ABB RobotStudio station: LATAM_caja_negra.rsstnx

Station Project3 (saved by RobotStudio 23.2.10395.0)
Controller IRB6640_130_320, task T_ROB1: task frame (RAPID world) sits at (1140.52, 0, 0) mm in the station
Controller IRB6640_130_320
  mechanical unit ROB_1: IRB6640_130_320__04, 6 joints, base frame (0, 0, 0) mm
Layout (positions relative to the parent item):
  - IRB6640_130_320__04 [mechanism, from %ABB.RobotStudio.Models.IRB6640%\IRB6640_130_320_G_04.rslib] at (1140.52, 0, 0) mm; joint values [0, 0, 0, 0, 0.1599, 0.0179] (rad or m)
  - Grupo_2 [graphiccomponentgroup]
    - Euro Pallet [graphiccomponentgroup, from Equipment\Euro Pallet.rslib] at (0, -2846.4, -3.2) mm
      - Body 1 [part, from Equipment\Euro Pallet.rslib]
    - Euro Pallet_2 [graphiccomponentgroup, from Equipment\Euro Pallet.rslib] at (0, -2029.21, -3.2) mm
      - Body 1 [part, from Equipment\Euro Pallet.rslib]
    - Euro Pallet_4 [graphiccomponentgroup, from Equipment\Euro Pallet.rslib] at (1157.68, -2846.4, -3.2) mm
      - Body 1 [part, from Equipment\Euro Pallet.rslib]
    - Euro Pallet_3 [graphiccomponentgroup, from Equipment\Euro Pallet.rslib] at (1157.68, -2029.21, -3.2) mm
      - Body 1 [part, from Equipment\Euro Pallet.rslib]
  - IRC5 [part, from %ABB.RobotStudio.Models.IRC5%\IRC5_Control-Module.rslib] at (5669.92, -980.14, 100) mm, rotated rx 90 ry 0 rz 90 deg
  - Pieza_2 [part] at (1194.52, -1963.54, 134.82) mm, size 600 x 600 x 200 mm
  - propeller [part, from Training Objects\propeller.rslib] at (625, 0, 373) mm, rotated rx 0 ry 0 rz 12 deg
  - IRB1200_5_90_STD_03 [mechanism, from %ABB.RobotStudio.Models.IRB1200%\IRB1200_5_90_STD_03.rslib] at (3914.45, 3690.17, 640.27) mm, rotated rx 0 ry 0 rz -177.61 deg; joint values [0, 0, 0, 0, 0.5236, 0] (rad or m)
  - Pieza_3 [part] at (3715.49, 3430.98, 0) mm, size 500 x 500 x 600 mm
  - Grupo_3 [graphiccomponentgroup]
    - Fence_2500_3 [graphiccomponentgroup, from Equipment\Fence_2500.rslib] at (-6063.8, 1734.17, 0) mm
      - Body 1 [part, from Equipment\Fence_2500.rslib]
      - Body 2 [part, from Equipment\Fence_2500.rslib]
    - Fence_2500_4 [graphiccomponentgroup, from Equipment\Fence_2500.rslib] at (-5999.52, 4213.05, 0) mm
      - Body 1 [part, from Equipment\Fence_2500.rslib]
      - Body 2 [part, from Equipment\Fence_2500.rslib]
    - Fence_2500_2 [graphiccomponentgroup, from Equipment\Fence_2500.rslib] at (-6042.58, -669.32, 0) mm
      - Body 1 [part, from Equipment\Fence_2500.rslib] at (0, -91.47, 0) mm
      - Body 2 [part, from Equipment\Fence_2500.rslib]
    - Fence_2500 [graphiccomponentgroup, from Equipment\Fence_2500.rslib] at (-5950.27, -3103.88, 0) mm
      - Body 1 [part, from Equipment\Fence_2500.rslib] at (0, -91.47, 0) mm
      - Body 2 [part, from Equipment\Fence_2500.rslib]
  - Grupo_4 [graphiccomponentgroup] at (10944.14, 0, 0) mm
    - Fence_2500_3 [graphiccomponentgroup, from Equipment\Fence_2500.rslib] at (-6063.8, 1734.17, 0) mm
      - Body 1 [part, from Equipment\Fence_2500.rslib]
      - Body 2 [part, from Equipment\Fence_2500.rslib]
    - Fence_2500_4 [graphiccomponentgroup, from Equipment\Fence_2500.rslib] at (-5999.52, 4213.05, 0) mm
      - Body 1 [part, from Equipment\Fence_2500.rslib]
      - Body 2 [part, from Equipment\Fence_2500.rslib]
    - Fence_2500_2 [graphiccomponentgroup, from Equipment\Fence_2500.rslib] at (-6042.58, -669.32, 0) mm
      - Body 1 [part, from Equipment\Fence_2500.rslib] at (0, -91.47, 0) mm
      - Body 2 [part, from Equipment\Fence_2500.rslib]
    - Fence_2500 [graphiccomponentgroup, from Equipment\Fence_2500.rslib] at (-5950.27, -3103.88, 0) mm
      - Body 1 [part, from Equipment\Fence_2500.rslib] at (0, -91.47, 0) mm
      - Body 2 [part, from Equipment\Fence_2500.rslib]
  - Grupo_5 [graphiccomponentgroup]
    - 950_4000_h2 [part, from %ABB.RobotStudio.Models.Conveyors%\Conveyor 950 4000 h2.rslib] at (3638.72, -1101.13, 242.49) mm, rotated rx 0 ry 0 rz 90.05 deg
    - 950_4000 [part, from %ABB.RobotStudio.Models.Conveyors%\Conveyor 950 4000 h2.rslib] at (3638.72, 3166.35, 242.49) mm, rotated rx 0 ry 0 rz 90.05 deg
  - Grupo_6 [graphiccomponentgroup] at (0, -9897.8, 0) mm
    - Fence_2500_11 [graphiccomponentgroup, from Equipment\Fence_2500.rslib] at (4938.96, 6750.42, 0) mm, rotated rx 0 ry 0 rz 90.25 deg
      - Body 1 [part, from Equipment\Fence_2500.rslib]
      - Body 2 [part, from Equipment\Fence_2500.rslib]
    - Fence_2500_9 [graphiccomponentgroup, from Equipment\Fence_2500.rslib] at (2444.62, 6739.42, 0) mm, rotated rx 0 ry 0 rz 90.25 deg
      - Body 1 [part, from Equipment\Fence_2500.rslib]
      - Body 2 [part, from Equipment\Fence_2500.rslib]
  - Grupo_7 [graphiccomponentgroup]
    - Fence_2500_11 [graphiccomponentgroup, from Equipment\Fence_2500.rslib] at (1507.61, 6735.29, 0) mm, rotated rx 0 ry 0 rz 90.25 deg
      - Body 1 [part, from Equipment\Fence_2500.rslib]
      - Body 2 [part, from Equipment\Fence_2500.rslib]
    - Fence_2500_10 [graphiccomponentgroup, from Equipment\Fence_2500.rslib] at (-3465.34, 6713.35, 0) mm, rotated rx 0 ry 0 rz 90.25 deg
      - Body 1 [part, from Equipment\Fence_2500.rslib]
      - Body 2 [part, from Equipment\Fence_2500.rslib]
    - Fence_2500_9 [graphiccomponentgroup, from Equipment\Fence_2500.rslib] at (-986.73, 6724.29, 0) mm, rotated rx 0 ry 0 rz 90.25 deg
      - Body 1 [part, from Equipment\Fence_2500.rslib]
      - Body 2 [part, from Equipment\Fence_2500.rslib]
    - Fence_740 [graphiccomponentgroup, from Equipment\Fence_740.rslib] at (4866.17, 6674.2, 0) mm, rotated rx 0 ry 0 rz 90.34 deg
      - Body 1 [part, from Equipment\Fence_740.rslib]
      - Body 2 [part, from Equipment\Fence_740.rslib]
Targets, tools, work objects and paths stored in the station, written as RAPID:
! task T_ROB1
MODULE CalibData
  PERS tooldata MyTool:=[TRUE,[[31.792631019,0,229.638935148],[0.945518576,0,0.325568154,0]],[1,[0,0,1],[1,0,0,0],0,0,0]];
ENDMODULE

